(*
Worker wrapper that runs different job each on iteration.
*)
FUNCTION_BLOCK LoopWorker
VAR
	_scheduler: Worker;
END_VAR

(*
Returns internal Worker.
*)
PROPERTY Base : I_Worker
GET
Base := _scheduler;
END_GET
END_PROPERTY

METHOD Run
VAR_INPUT
END_VAR
IF _scheduler.First = 0 THEN
	RETURN;
END_IF

CASE _scheduler.First.State OF
	JobState.Completed, JobState.Aborted:
		_scheduler.Dequeue(_scheduler.First);
END_CASE

CASE _scheduler.Run(_scheduler.First) OF
	Ok:
		_scheduler.Defer(_scheduler.First);
	Err.Itf0:
		RETURN;
	ELSE
		NewDebug(_scheduler, Param.EXE_INTERNAL_DEBUG_MODE, 'Scheduler: Incorrect task state!', _scheduler.First);
		RETURN;	
END_CASE
END_METHOD

END_FUNCTION_BLOCK

(* stored: Version 1.1.0.1
   POU LoopWorker: Id {441fb644-9147-45db-9af7-51cecc3c1e57}, SpecialFunc None
   Property Base: Id {177ef07f-71b2-407c-8753-27a70af21e29}
   Get Get: Id {585f641f-8de4-451e-807b-7a59f5f29825}
   Method Run: Id {f543f0f7-b0a8-4b9e-9878-1b8fa71dc1f9} *)
